(* PLC project GVL_PLC.generated, Beckhoff Automation GmbH TwinCAT PLC Control 3.5.13.21 *)
(* stored: creationDateTime 2026-05-28T16:52:01.2730334, modificationDateTime 2026-05-28T16:52:01.2730334 *)

TYPE stControl :
STRUCT
	{attribute 'OPC.UA.DA' := '1'}
	TargetValue : LREAL;
	{attribute 'OPC.UA.DA' := '1'}
	Unit : STRING;
	{attribute 'OPC.UA.DA' := '1'}
	SerialNumber : STRING;
END_STRUCT
END_TYPE

TYPE stMeasure :
STRUCT
	{attribute 'OPC.UA.DA' := '1'}
	ActualValue : LREAL;
	{attribute 'OPC.UA.DA' := '1'}
	Unit : STRING;
	{attribute 'OPC.UA.DA' := '1'}
	SerialNumber : STRING;
END_STRUCT
END_TYPE

TYPE stRingBuffer :
STRUCT
	{attribute 'OPC.UA.DA' := '1'}
	Buffer : ARRAY[1..4096] OF BYTE;
	{attribute 'OPC.UA.DA' := '1'}
	RdIdx : UINT;
	{attribute 'OPC.UA.DA' := '1'}
	WrIdx : UINT;
	{attribute 'OPC.UA.DA' := '1'}
	BufferSize : UINT := 4096;
END_STRUCT
END_TYPE

TYPE stSerialConfiguration :
STRUCT
	{attribute 'OPC.UA.DA' := '1'}
	BaudRate : UDINT := 57600;
	{attribute 'OPC.UA.DA' := '1'}
	Parity : INT := 0;
	{attribute 'OPC.UA.DA' := '1'}
	DataBits : INT := 8;
	{attribute 'OPC.UA.DA' := '1'}
	StopBits : INT := 1;
	{attribute 'OPC.UA.DA' := '1'}
	DTR : BOOL := FALSE;
	{attribute 'OPC.UA.DA' := '1'}
	RTS : BOOL := FALSE;
END_STRUCT
END_TYPE

TYPE stSerialConnection :
STRUCT
	{attribute 'OPC.UA.DA' := '1'}
	TxBuffer : stRingBuffer;
	{attribute 'OPC.UA.DA' := '1'}
	RxBuffer : stRingBuffer;
	{attribute 'OPC.UA.DA' := '1'}
	Reset : BOOL := TRUE;
	{attribute 'OPC.UA.DA' := '1'}
	ResetAck : BOOL;
	{attribute 'OPC.UA.DA' := '1'}
	Configuration : stSerialConfiguration;
	{attribute 'OPC.UA.DA' := '1'}
	TxError : ComError_t;
	{attribute 'OPC.UA.DA' := '1'}
	RxError : ComError_t;
END_STRUCT
END_TYPE

TYPE stSerialInternal :
STRUCT
	{attribute 'OPC.UA.DA' := '1'}
	RxBuffer : ComBuffer;
	{attribute 'OPC.UA.DA' := '1'}
	TxBuffer : ComBuffer;
	{attribute 'OPC.UA.DA' := '1'}
	CtrlError : BOOL;
	{attribute 'OPC.UA.DA' := '1'}
	CtrlErrorID : ComError_t;
END_STRUCT
END_TYPE

TYPE stPressureSource :
STRUCT
	{attribute 'OPC.UA.DA' := '1'}
	ActualValue : LREAL;
	{attribute 'OPC.UA.DA' := '1'}
	Unit : STRING;
	{attribute 'OPC.UA.DA' := '1'}
	SerialNumber : STRING;
END_STRUCT
END_TYPE

TYPE stTemperatureSource :
STRUCT
	{attribute 'OPC.UA.DA' := '1'}
	ActualValue : LREAL;
	{attribute 'OPC.UA.DA' := '1'}
	Unit : STRING;
	{attribute 'OPC.UA.DA' := '1'}
	SerialNumber : STRING;
END_STRUCT
END_TYPE

TYPE stMeasureWithZero EXTENDS stMeasure :
STRUCT
	{attribute 'OPC.UA.DA' := '1'}
	Zero : BOOL;
END_STRUCT
END_TYPE

CONFIGURATION Application
  RESOURCE GVL_PLC.generated ON PLC
(* global variable list GVL_PLC *)
{attribute 'qualified_only'}
VAR_GLOBAL
	{attribute 'OPC.UA.DA' := '1'}
	SystemStatus : UINT;
	{attribute 'OPC.UA.DA' := '1'}
	AllPartitiantsPresent : BOOL;
	{attribute 'OPC.UA.DA' := '1'}
	CANOpenState : BOOL;
	{attribute 'OPC.UA.DA' := '1'}
	IOLinkState : BOOL;
	{attribute 'OPC.UA.DA' := '1'}
	AppTimestamp : DT;
	{attribute 'OPC.UA.DA' := '1'}
	AppVersion : STRING;
END_VAR
VAR_GLOBAL CONSTANT
	iExpectedNumberOfPartitiants : UINT := 14;
END_VAR
(* global variable list GVL_Power *)
{attribute 'qualified_only'}
VAR_GLOBAL
	{attribute 'OPC.UA.DA' := '1'}
	SupplyVoltage24V_1 : LREAL;
	{attribute 'OPC.UA.DA' := '1'}
	SupplyVoltage24V_2 : LREAL;
	{attribute 'OPC.UA.DA' := '1'}
	SupplyVoltage24V_3 : LREAL;
	{attribute 'OPC.UA.DA' := '1'}
	SupplyVoltage24V_4 : LREAL;
	{attribute 'OPC.UA.DA' := '1'}
	SwitchSupplyPower_UUT : BOOL;
END_VAR
(* global variable list GVL_Pressure *)
{attribute 'qualified_only'}
VAR_GLOBAL
	{attribute 'OPC.UA.DA' := '1'}
	SystemPressureAtValveCluster : stMeasure;
	{attribute 'OPC.UA.DA' := '1'}
	SystemPressurePressureRegulator : stMeasure;
	{attribute 'OPC.UA.DA' := '1'}
	RelativePressure : ARRAY[1..1] OF stMeasureWithZero;
	{attribute 'OPC.UA.DA' := '1'}
	PressureRegulator : ARRAY[1..1] OF stControl;
END_VAR
VAR_GLOBAL CONSTANT
	NumberOfWika : INT := 1;
	NumberOfRegulator : INT := 1;
END_VAR
(* global variable list GVL_Resistance *)
{attribute 'qualified_only'}
VAR_GLOBAL
	{attribute 'OPC.UA.DA' := '1'}
	FunctionalEarthUUT : LREAL;
	{attribute 'OPC.UA.DA' := '1'}
	FunctionalEarthUUTOverrange : BOOL;
	{attribute 'OPC.UA.DA' := '1'}
	FunctionalEarthUUTUnderrange : BOOL;
END_VAR
(* global variable list GVL_Serial *)
{attribute 'qualified_only'}
VAR_GLOBAL
	{attribute 'OPC.UA.DA' := '1'}
	SerialControl : ARRAY[1..1] OF stSerialInternal;
	{attribute 'OPC.UA.DA' := '1'}
	SerialConnections : ARRAY[1..1] OF stSerialConnection;
END_VAR
VAR_GLOBAL CONSTANT
	iNumberOfSerial : INT := 1;
	aSerialConnectionSide : ARRAY[1..1] OF INT;
END_VAR
(* global variable list GVL_Status *)
{attribute 'qualified_only'}
VAR_GLOBAL
	{attribute 'OPC.UA.DA' := '1'}
	Green : BOOL;
	{attribute 'OPC.UA.DA' := '1'}
	Yellow : BOOL;
	{attribute 'OPC.UA.DA' := '1'}
	Red : BOOL;
	{attribute 'OPC.UA.DA' := '1'}
	Blue : BOOL;
	{attribute 'OPC.UA.DA' := '1'}
	White : BOOL;
	{attribute 'OPC.UA.DA' := '1'}
	IsDutAdapted : BOOL;
	{attribute 'OPC.UA.DA' := '1'}
	SwitchDockSignal_UUT : BOOL;
END_VAR
(* global variable list GVL_Temperature *)
{attribute 'qualified_only'}
VAR_GLOBAL
	{attribute 'OPC.UA.DA' := '1'}
	TemperatureSensor : ARRAY[1..1] OF stTemperatureSource;
END_VAR
VAR_GLOBAL CONSTANT
	maxTemperatureSensorCount : INT := 1;
END_VAR
(* global variable list GVL_Valves *)
{attribute 'qualified_only'}
VAR_GLOBAL
	{attribute 'OPC.UA.DA' := '1'}
	P1 : ARRAY[1..16] OF BOOL;
	{attribute 'OPC.UA.DA' := '1'}
	V12 : BOOL;
	{attribute 'OPC.UA.DA' := '1'}
	V12_cyclic : BOOL := FALSE;
	{attribute 'OPC.UA.DA' := '1'}
	V12_onTime : INT := 5000;
	{attribute 'OPC.UA.DA' := '1'}
	V12_offTime : INT := 5000;
END_VAR
VAR_GLOBAL CONSTANT
	minValveCount : INT := 1;
	maxValveCount : INT := 16;
END_VAR
(* global variable list Global_Version *)
{attribute 'qualified_only'}
VAR_GLOBAL CONSTANT
	stLibVersion_A220053_Vapor_5000_Function_Test : ST_LibVersion;
END_VAR
    TASK PlcTask(INTERVAL := T#0ms, PRIORITY := 20);
    TASK PlcTask1ms(INTERVAL := T#0ms, PRIORITY := 4);
    PROGRAM MAIN WITH PlcTask : MAIN;
    PROGRAM Background WITH PlcTask1ms : Background;
  END_RESOURCE
END_CONFIGURATION
